TYPE
    U_ProfinetDeviceDiagInput :
    UNION
        uUint  : UINT;
        aBytes : ARRAY[0..1] OF BYTE;
    END_UNION
END_TYPE

(* stored: Version 1.1.0.1, ProductVersion 3.1.4024.12
   DUT U_ProfinetDeviceDiagInput: Id {68644c1f-f362-4e13-bd82-1b67d26c626f} *)
